TYPE ST_PumpGrundfosMagna3DefaultParameters :
STRUCT
	bExternalTemperatureSensor 	: BOOL := TRUE;
	bPumpBeforeApplication : BOOL := TRUE;
	fControllerAmplification : LREAL := 0.265;
	tControllerIntegralTime : TIME := T#15S;
	tTaskCycleTime	: TIME := GlobalVariables.tTaskCycleTime_MAIN;
	tCtrlCycleTime	: TIME := GlobalVariables.tCtrlCycleTime_MAIN;	
	aSetPointLimits	: ARRAY[1..2] OF REAL := [0,100];
END_STRUCT
END_TYPE

(* stored: Version 1.1.0.1, ProductVersion 3.1.4024.10
   DUT ST_PumpGrundfosMagna3DefaultParameters: Id {c79135d6-6136-4193-87e6-f0a4d4d2cc36} *)
